// TIA Portal V19 export
DATA_BLOCK "ControlNodes"   // DB62
// stored: Access Published, MemoryReserve 100, Namespace Unit2.EM1
   VAR
      em { ExternalWritable := 'False'} : "LAF_typeEmControlNode";
      jobs { ExternalWritable := 'False'} : "LAF_typeJobs";
      sequence { ExternalWritable := 'False'} : "LAF_typeSequence";
      cm1Vfd205 : "LEXCHANGETRAY_typeRollerVfdContronNode";
      cm2SingalTM { S7_SetPoint := 'True'} : "LEXCHANGETRAY_typeRollerIoSignalControlNode";
   END_VAR
BEGIN
   em.status.enabled := true;
END_DATA_BLOCK
